PROGRAM MAIN
VAR
	axisCtrls : ARRAY[1 .. 10] OF AxisCtrl;
	i : INT := 0;
	
END_VAR

FOR i := 1 TO 10 DO
 	axisCtrls[i]();
END_FOR;

END_PROGRAM

(* stored: Version 1.1.0.1, ProductVersion 3.1.4020.12
   POU MAIN: Id {0196f569-7f4c-4cc8-b953-20d0a877f80a}, SpecialFunc None *)
